{attribute 'qualified_only'}
{attribute 'to_string'}
TYPE ZAppStep :
(
  Undefined := 0
  
  ,BootBegin
  ,BootLoadDefaultData
  ,BootEnd
  ,BootFaultBegin
  ,BootFaultEnd 
  ,RunningBegin
  ,RunningEnd   
);
END_TYPE

(* stored: Version 1.1.0.1
   DUT ZAppStep: Id {92fb12a7-4de8-44b2-8f09-03a5516ba197} *)
